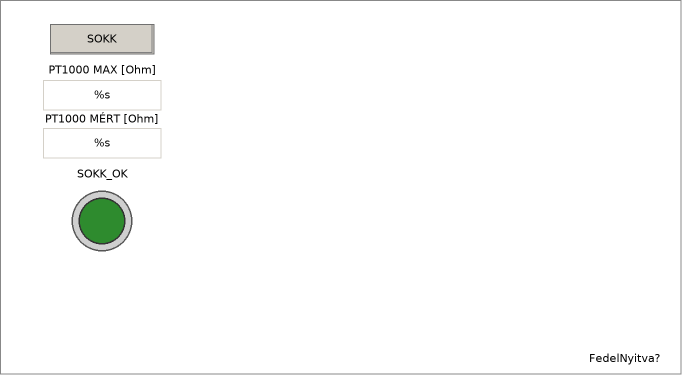
VISUALIZATION Vegmero_sokk  // 682x375
    Label (570,344 110x29), "FedelNyitva?"
    Textfield (43,128 118x30), "%s", text variable: VEGMERO.rPTRES
    Textfield (43,80 118x30), "%s", text variable: GVL.PTRES_SOKK_MAX
    Label (35,109 134x20), "PT1000 MÉRT [Ohm]"
    Label (39,60 127x20), "PT1000 MAX [Ohm]"
    Button (50,24 104x30), "SOKK", input disabled if: VEGMERO.s_InCommand<>''
        OnMouseUp: execute { VEGMERO.s_InCommand:='SOKK'; }
    Lamp1 (67,186 70x70), variable: NOT GVL.bShockOK, style: Lamp-Lamp1-Red
    Label (70,164 65x20), "SOKK_OK"
    Lamp1 (67,186 70x70), variable: GVL.bShockOK, invisible if: NOT GVL.bShockOK AND VEGMERO.bSOKK_MERVE, style: Lamp-Lamp1-Green
END_VISUALIZATION

(* stored: Version 1.1.0.1, ProductVersion 3.1.4024.11
   Visu Vegmero_sokk: Id {0b4ca247-3e5b-4037-bca6-ed624fd2de05} *)
